// TIA Portal V18 export
DATA_BLOCK "HMI ALARM DB"   // DB5
{ S7_Optimized_Access := 'FALSE' }
VERSION : 0.1
// stored: AutoNumber true, DBAccessibleFromOPCUA true, IsOnlyStoredInLoadMemory false, IsWriteProtectedInAS false
   VAR
      "FEED PUMP" : Byte;   // XO- INTERLOCK
      "ACID DOSING" : Byte;   // X1 - TRIP
      "CAUSTIC DOSING" : Byte;   // X2 - RUN FB ERROR
      "RP 1" : Byte;
      "RP 2" : Byte;
      "RP 3" : Byte;
      "RETURN NOT SELECTED" : Bool;
      "CYCLE NOT SELECTED" : Bool;
      "WATER FLUSH TIME NOT SET" : Bool;
      "HOT WATER TIME NOT SET" : Bool;
      "RECUP TIME NOT SET" : Bool;
      "ACIDIC TIME NOT SET" : Bool;
      "CAUSTIC TIMENOT SET" : Bool;
   END_VAR
BEGIN
END_DATA_BLOCK
